Staubli VAL3: _moveToScan.pgx

program _moveToScan()
begin
  // ============================================================================
  // CMD 2: 스캔 위치로 이동
  // ============================================================================
  cls()
  putln("[CMD "+ toString("", nCmdSignal) +"] 스캔 위치로 이동")
  nStatusSignal = 0

  movej(j_scan, tTool, mNomSpeed)
  waitEndMove()

  putln("[CMD 2] 완료 - STATUS=1")
  nStatusSignal = 1

end
